// TwinCAT 3 PLC project PLCStudent
// ProgramVersion: 3.1.4024.0
// libraries:
//   Tc2_Standard, * (Beckhoff Automation GmbH)
//   Tc2_System, * (Beckhoff Automation GmbH)
//   Tc3_Module, * (Beckhoff Automation GmbH)
// project tree:
//   / GlobalTextList.TcGTLO, PlcTask.TcTTO, Visualization Manager.TcVMO (not stored)
//   GVLs/ GVL.TcGVL
//   POUs/ Automatic.TcPOU, Automatic_Or_Manual.TcPOU, Emergency_Stop.TcPOU, MAIN.TcPOU, Manual.TcPOU, Stop.TcPOU
//   VISUs/ HMI.TcVIS
// (motion and I/O tree: see PLC project plcsim)
// real-time tasks:
//   TASK PlcTask: cycle T#10ms, priority 20, ADS port 350
//   TASK PlcTask1: cycle T#10ms, priority 21, ADS port 351
// variable links:
//   PLCSim/PLCSim Instance <-> PLCStudent/PLCStudent Instance
//     PlcTask Inputs/GVL.ixGotoPosA <-> PlcTask Outputs/GVL.qxGotoPosA
//     PlcTask Inputs/GVL.ixGotoPosB <-> PlcTask Outputs/GVL.qxGotoPosB
//     PlcTask Outputs/GVL.qxA <-> PlcTask Inputs/GVL.ixA
//     PlcTask Outputs/GVL.qxB <-> PlcTask Inputs/GVL.ixB
//     PlcTask Outputs/GVL.qxTram <-> PlcTask Inputs/GVL.ixTram

CONFIGURATION PLCStudent
    RESOURCE PLC ON TwinCAT3
        TASK PlcTask(INTERVAL := T#10ms, PRIORITY := 21);
        PROGRAM MAIN WITH PlcTask : MAIN;
    END_RESOURCE
END_CONFIGURATION

// ---- GVLs/GVL.TcGVL
{attribute 'qualified_only'}
VAR_GLOBAL
	//Output from process
	ixTram	AT %I*: BOOL;
	ixA		AT %I*: BOOL;
	ixB		AT %I*: BOOL;
	
	//Input to from Operator
	qxGotoPosB AT %Q*: BOOL;
	qxGotoPosA AT %Q*: BOOL;
	//qcStop AT %I*: BOOL;
	//qxEmergency AT %I*: BOOL;
END_VAR

// ---- POUs/MAIN.TcPOU
PROGRAM MAIN
VAR
	Manual_Automatic:BOOL;
	Visible:BOOL;
END_VAR

Stop();
Emergency_Stop();
Automatic_Or_Manual();
Visible:=not gvl.ixA;

END_PROGRAM

// ---- POUs/Stop.TcPOU
PROGRAM Stop
VAR
	Stop_Button:BOOL;
	Break_At_Home: BOOL;
END_VAR

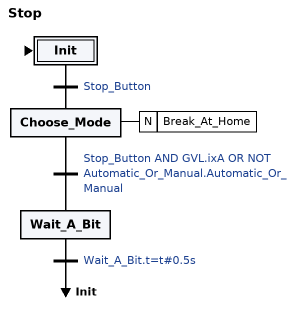
INITIAL_STEP Init:
END_STEP
TRANSITION FROM Init TO Choose_Mode
    := Stop_Button;
END_TRANSITION
STEP Choose_Mode:
    Break_At_Home(N);
END_STEP
TRANSITION FROM Choose_Mode TO Wait_A_Bit
    := Stop_Button AND GVL.ixA OR NOT Automatic_Or_Manual.Automatic_Or_Manual;
END_TRANSITION
STEP Wait_A_Bit:
END_STEP
TRANSITION FROM Wait_A_Bit TO Init
    := Wait_A_Bit.t=t#0.5s;
END_TRANSITION

END_PROGRAM

// ---- POUs/Automatic_Or_Manual.TcPOU
PROGRAM Automatic_Or_Manual
VAR_INPUT
	Automatic_Or_Manual:BOOL;
END_VAR

IF Automatic_Or_Manual THEN
	Automatic();
ELSE
	Manual();
END_IF

END_PROGRAM

// ---- POUs/Automatic.TcPOU
PROGRAM Automatic
VAR
END_VAR

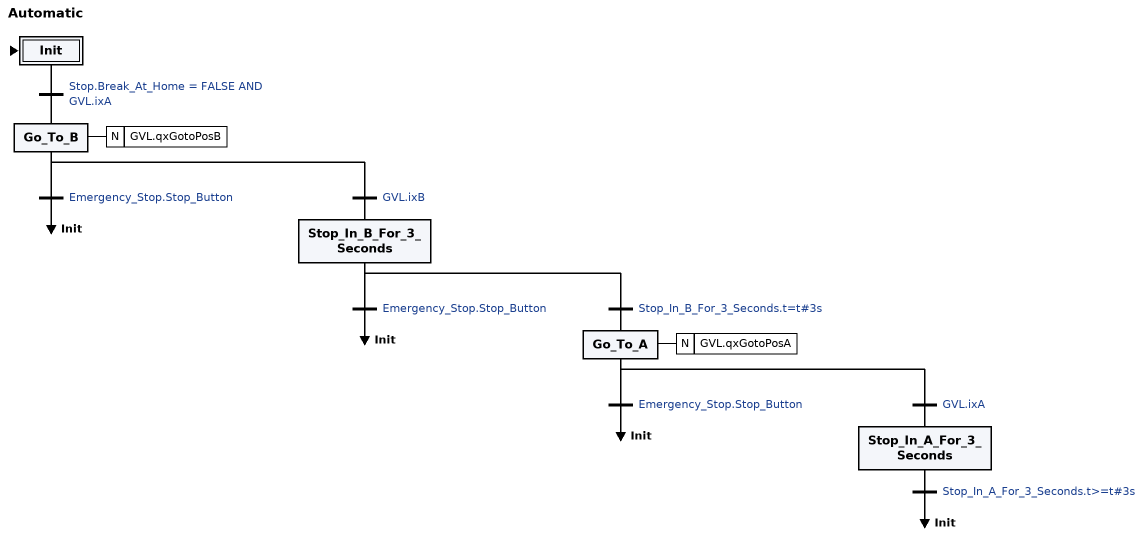
INITIAL_STEP Init:
END_STEP
TRANSITION FROM Init TO Go_To_B
    := Stop.Break_At_Home = FALSE AND GVL.ixA;
END_TRANSITION
STEP Go_To_B:
    GVL.qxGotoPosB(N);
END_STEP
TRANSITION FROM Go_To_B TO Init
    := Emergency_Stop.Stop_Button;
END_TRANSITION
TRANSITION FROM Go_To_B TO Stop_In_B_For_3_Seconds
    := GVL.ixB;
END_TRANSITION
STEP Stop_In_B_For_3_Seconds:
END_STEP
TRANSITION FROM Stop_In_B_For_3_Seconds TO Init
    := Emergency_Stop.Stop_Button;
END_TRANSITION
TRANSITION FROM Stop_In_B_For_3_Seconds TO Go_To_A
    := Stop_In_B_For_3_Seconds.t=t#3s;
END_TRANSITION
STEP Go_To_A:
    GVL.qxGotoPosA(N);
END_STEP
TRANSITION FROM Go_To_A TO Init
    := Emergency_Stop.Stop_Button;
END_TRANSITION
TRANSITION FROM Go_To_A TO Stop_In_A_For_3_Seconds
    := GVL.ixA;
END_TRANSITION
STEP Stop_In_A_For_3_Seconds:
END_STEP
TRANSITION FROM Stop_In_A_For_3_Seconds TO Init
    := Stop_In_A_For_3_Seconds.t>=t#3s;
END_TRANSITION

END_PROGRAM

// ---- POUs/Emergency_Stop.TcPOU
PROGRAM Emergency_Stop
VAR
	Stop_Button:BOOL;
END_VAR

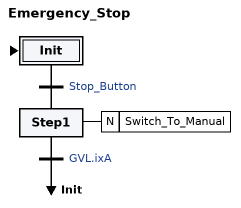
INITIAL_STEP Init:
END_STEP
TRANSITION FROM Init TO Step1
    := Stop_Button;
END_TRANSITION
STEP Step1:
    Switch_To_Manual(N);
END_STEP
TRANSITION FROM Step1 TO Init
    := GVL.ixA;
END_TRANSITION

ACTION Switch_To_Manual:
Automatic_Or_Manual.Automatic_Or_Manual:=FALSE;
END_ACTION

END_PROGRAM

// ---- POUs/Manual.TcPOU
PROGRAM Manual
VAR
	Left:BOOL;
	Right:BOOL;
END_VAR

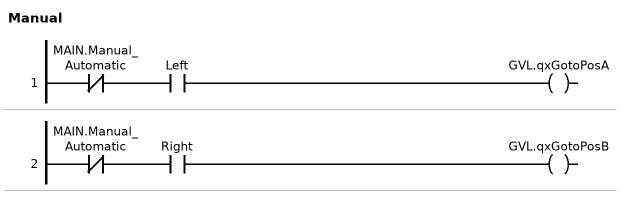
// NETWORK 1
GVL.qxGotoPosA := NOT MAIN.Manual_Automatic AND Left;

// NETWORK 2
GVL.qxGotoPosB := NOT MAIN.Manual_Automatic AND Right;

END_PROGRAM

// ---- GlobalTextList.TcGTLO
TEXTLIST GlobalTextList
  195 = 'Emergency stop'
  775 = 'Left'
  813 = 'Right'
  168 = 'Stop'
END_TEXTLIST

// ---- VISUs/HMI.TcVIS
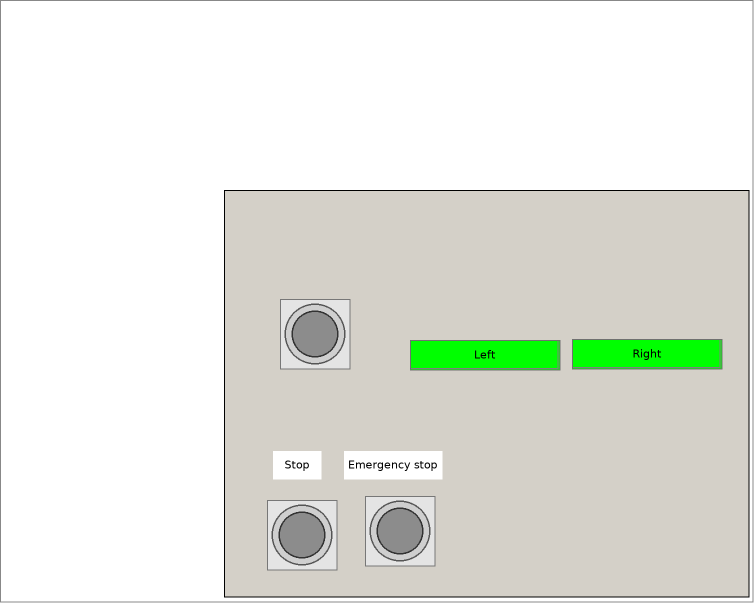
VISUALIZATION HMI  // 754x603
    Rectangle (224,190 525x407)
    Polyline (573,328)
    PushSwitch (267,500 70x70), variable: Stop.Stop_Button, behaviour: TAP, style: Switch-PushSwitch-Gray
    PushSwitch (365,496 70x70), variable: Emergency_Stop.Stop_Button, behaviour: TAP, style: Switch-PushSwitch-Gray
    Button (410,340 150x30), "Left", colour toggle: GVL.qxGotoPosA
        tap Manual.Left
    Button (572,339 150x30), "Right", colour toggle: GVL.qxGotoPosB
        tap Manual.Right
    Textfield (272,450 50x30), "Stop"
    Textfield (343,450 100x30), "Emergency stop"
    PushSwitchLed (280,299 70x70), variable: Automatic_Or_Manual.Automatic_Or_Manual, invisible if: MAIN.Visible, behaviour: TOGGLE, style: Switch-PushSwitchLed-Gray
END_VISUALIZATION
